
// ===== library: MasterCopy "myDataType" =====

TYPE "myDataType"
   STRUCT
      myStruct : Struct
         "Int" : Int;
         "Bool" : Bool;
      END_STRUCT;
   END_STRUCT;
END_TYPE

// ===== library: MasterCopy "Block_1" =====

FUNCTION_BLOCK "Block_1"   // FB3, SCL
{ S7_Optimized_Access := 'TRUE' }
VERSION : 0.1
   VAR_INPUT
      "Time" : Time;
   END_VAR
BEGIN
END_FUNCTION_BLOCK

// ===== library: MasterCopy "MAC_use_casesFB" =====

// folder: Libraries/Lib_MAC_use_cases_Blocks

FUNCTION_BLOCK "MAC_use_casesFB"   // FB4, FBD
TITLE = BasicFB
{ S7_Optimized_Access := 'TRUE' }
VERSION : 0.1
   VAR_INPUT
      Input1 : Bool;
      Input2 : Bool;
   END_VAR
   VAR_OUTPUT
      Time_output1 : Time;
      Output1 : Bool;
   END_VAR
BEGIN

REGION Network 1: AndNetwork1
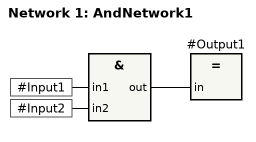
   #Output1 := #Input1 AND #Input2;
END_REGION
END_FUNCTION_BLOCK

// ===== library: MasterCopy "MAC_use_casesFB_FailSafe" =====

// folder: Libraries/Lib_MAC_use_cases_Blocks

FUNCTION_BLOCK "MAC_use_casesFB_FailSafe"   // FB8, F_FBD
TITLE = FailSafe FB
{ S7_Optimized_Access := 'TRUE' }
VERSION : 0.1
   VAR_INPUT
      Input1 : Bool;
      Input2 : Bool;
   END_VAR
   VAR_OUTPUT
      Time_output1 : Time;
      Output1 : Bool;
   END_VAR
BEGIN

REGION Network 1: AndNetwork1
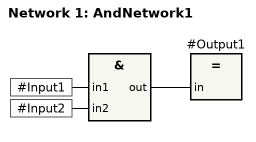
   #Output1 := #Input1 AND #Input2;
END_REGION
END_FUNCTION_BLOCK